FUNCTION_BLOCK E_CTUD (* Event-Driven Up-Down Counter *)
  (* Standard: 61499-1-A.x; Classification: Event-driven blocks; Function: Up-Down-counter; Description: Copyright (c) 2017 fortiss GmbH 2019 Johannes Keppler University Linz This program and the accompanying materials are made available under the terms of the Eclipse Public License 2.0 which is available at https://www.eclipse.org/legal/epl-2.0/ SPDX-License-Identifier: EPL-2.0 *)
  (* Version 3.0, 2025-04-14, Franz H??pfinger, HR Agrartechnik GmbH, Made Version 3.0.0 inspired by Work from Patrick Aigner *)
  (* Version 1.1, 2019-07-09, Alois Zoitl, JKU, fixed bug in down counting *)
  (* Version 1.0, 2017-09-22, Alois Zoitl, fortiss GmbH, initial API and implementation and/or initial documentation *)
  PACKAGE iec61499::events;
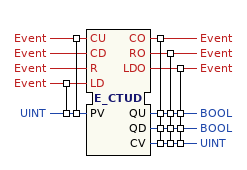
  EVENT_INPUT
    CU WITH PV; (* Count Up *)
    CD; (* Count Down *)
    R; (* Reset *)
    LD WITH PV; (* Load *)
  END_EVENT
  EVENT_OUTPUT
    CO WITH QU, CV, QD; (* Count Output Event *)
    RO WITH QU, CV, QD; (* Reset Output Event *)
    LDO WITH QU, QD, CV;
  END_EVENT
  VAR_INPUT
    PV : UINT; (* Preset Value *)
  END_VAR
  VAR_OUTPUT
    QU : BOOL; (* CV >=PV *)
    QD : BOOL; (* CV <= 0 *)
    CV : UINT; (* Counter Value *)
  END_VAR
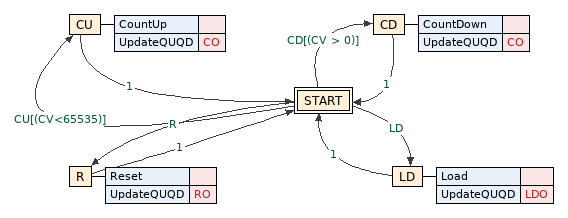
  EC_STATES
    START;
    CU : CountUp, UpdateQUQD -> CO;
    R : Reset, UpdateQUQD -> RO;
    CD : CountDown, UpdateQUQD -> CO;
    LD : Load, UpdateQUQD -> LDO;
  END_STATES
  EC_TRANSITIONS
    START TO CU := CU[(CV<65535)];
    CU TO START := 1;
    START TO R := R;
    R TO START := 1;
    START TO CD := CD[(CV > 0)];
    CD TO START := 1;
    START TO LD := LD;
    LD TO START := 1;
  END_TRANSITIONS
  ALGORITHM CountUp IN ST: (* Count Up *)
CV := CV + 1;
  END_ALGORITHM
  ALGORITHM Reset IN ST: (* Reset *)
CV := 0;
  END_ALGORITHM
  ALGORITHM Load IN ST: (* ALG *)
CV := PV;
  END_ALGORITHM
  ALGORITHM UpdateQUQD IN ST: (* ALG *)
QU := (CV>= PV);
QD := (CV = 0);
  END_ALGORITHM
  ALGORITHM CountDown IN ST: (* ALG *)
CV := CV - 1;
  END_ALGORITHM
END_FUNCTION_BLOCK
